# EPICS substitutions: apps/ftIntlkApp/Db/prad-gems-intlk.substitutions
file "db/mmIntlk.template" {
pattern { P R PV LOW HIGH CTRL CTRLVAL PREC DESC }
{ B_DET_PRADGEM_INTLK_ GasFlt            B_DET_PRADGEM_GAS_FLT               -99999                                  1                                       B_DET_PRADGEM_HV:OFF 1 0 "Turn HV OFF if PLC fault" }
{ B_DET_PRADGEM_INTLK_ GasPress          B_DET_PRADGEM_GAS_MIX1_PRESS        B_DET_PRADGEM_GAS_MIX1_PRESS.LOLO       B_DET_PRADGEM_GAS_MIX1_PRESS.HIHI       B_DET_PRADGEM_HV:OFF 1 2 "Turn HV OFF if Mix1 pressure LOLO/HIHI" }
{ B_DET_PRADGEM_INTLK_ GasInflowHi       B_DET_PRADGEM_GAS_INFLOW            -99999                                  B_DET_PRADGEM_GAS_INFLOW.HIHI           B_DET_PRADGEM_HV:OFF 1 2 "Turn HV OFF if inflow HIHI" }
{ B_DET_PRADGEM_INTLK_ GasInflowLo       B_DET_PRADGEM_GAS_INFLOW            0.3                                     999999                                  B_DET_PRADGEM_HV:OFF 1 2 "Turn HV OFF if inflow < 0.3" }
{ B_DET_PRADGEM_INTLK_ GasArFlowFrac     B_DET_MVT_GAS_MIX1_Ar_FLOW_FRAC     B_DET_MVT_GAS_MIX1_Ar_FLOW_FRAC.LOLO    B_DET_MVT_GAS_MIX1_Ar_FLOW_FRAC.HIHI    B_DET_PRADGEM_HV:OFF 1 2 "Turn HV OFF if Argon flow LOLO/HIHI" }
{ B_DET_PRADGEM_INTLK_ GasC4H10FlowFrac  B_DET_MVT_GAS_MIX1_C4H10_FLOW_FRAC  B_DET_MVT_GAS_MIX1_C4H10_FLOW_FRAC.LOLO B_DET_MVT_GAS_MIX1_C4H10_FLOW_FRAC.HIHI B_DET_PRADGEM_HV:OFF 1 2 "Turn HV OFF if C4H10 flow LOLO/HIHI" }
}
